TYPE ST_MasterboardData :
STRUCT
	// Masterboard Data (Value 3)
	MasterboardData: ARRAY [1..74] OF BYTE;

END_STRUCT
END_TYPE

(* stored: Version 1.1.0.1, ProductVersion 3.1.4020.12
   DUT ST_MasterboardData: Id {0a4a6a29-b039-41bd-991b-672596544d26} *)
